// TIA Portal V20 export
DATA_BLOCK "DB_GestionWorkingModes"   // DB132
// stored: InstanceOfName FB_GestionWorkingModes, InstanceOfType FB
"FB_GestionWorkingModes"
   // VAR
   //    sMCP_KxxKeysDisable : Bool;
   // END_VAR
BEGIN
END_DATA_BLOCK
